VAR_GLOBAL CONSTANT
	cuintMaxStation: INT := 4;
END_VAR

(* stored: Version 1.1.0.1, ProductVersion 3.1.0.23
   GVL Const_HFE: Id {dff3989f-620a-4448-99a3-71d687dfd026} *)
